// TwinCAT 3 PLC project unit_tests
// ProgramVersion: 3.1.4024.0
// libraries:
//   Tc2_Standard, * (Beckhoff Automation GmbH)
//   Tc2_System, * (Beckhoff Automation GmbH)
//   Tc3_Module, * (Beckhoff Automation GmbH)
//   TcUnit, * (www.tcunit.org)
// project tree:
//   / UnitTests.TcTTO, UNIT_TESTS.TcPOU

CONFIGURATION unit_tests
    RESOURCE PLC ON TwinCAT3
        TASK UnitTests(INTERVAL := T#10ms, PRIORITY := 1);
        PROGRAM UNIT_TESTS WITH UnitTests : UNIT_TESTS;
    END_RESOURCE
END_CONFIGURATION

// ---- UNIT_TESTS.TcPOU
PROGRAM UNIT_TESTS
VAR

END_VAR

TcUnit.RUN_IN_SEQUENCE();

END_PROGRAM
